Staubli VAL3: numCopy.pgx

public program numCopy(num& x_nCopy[] (dimensions=1), num& x_nPaste[] (dimensions=1))
// Copy all the value from the x_nCopy to x_nPaste
  local num i
  local num l_nSize
begin
  // Copy all the value from the first element to the second one
  //
  // redim the Paste String ARRAY
  //
  l_nSize=size(x_nPaste)
  if size(x_nCopy)>size(x_nPaste)
    for i=l_nSize to (size(x_nCopy)-1)
      insert(x_nPaste[i])
    endFor
  else
    if size(x_nCopy)<size(x_nPaste)
      for i=size(x_nCopy) to l_nSize-1
        delete(x_nPaste[size(x_nCopy)])
      endFor
    endIf
  endIf
  // COPY ALL THE FIELD
  for i=0 to (size(x_nCopy)-1)
    x_nPaste[i]=x_nCopy[i]
  endFor
end
